// TIA Portal V17 export
// export: Created 2022-07-16T16:56:13.7076572Z, ExportSetting WithDefaults, DisplayName Totally Integrated Automation Portal, DisplayVersion V17, DisplayName TIA Portal Openness, DisplayVersion V17, DisplayName TIA Portal Version Control Interface, DisplayVersion V17, DisplayName TIA Portal Test Suite Advanced, DisplayVersion V17, DisplayName STEP 7 Professional, DisplayVersion V17, DisplayName STEP 7 Safety, DisplayVersion V17, DisplayName WinCC Professional, DisplayVersion V17
TYPE "Client interface_1.dbData.postTestResult.preTestCheckSequence.pressures.airHoldTest"
// stored: IsFailsafeCompliant false
   STRUCT
      preDwellPeriod { ExternalWritable := 'False'} : Bool;
      postDwellPeriod { ExternalWritable := 'False'} : Bool;
   END_STRUCT;
END_TYPE
